// TwinCAT 3 PLC project ServerMappingSampleProject_PLC2
// Title: TF6100_OpcUa_Server_Sample_PLC2
// Company: Beckhoff Automation Gmbh
// ProjectVersion: 0.0.0.0
// ProgramVersion: 3.1.4026.17
// libraries:
//   Tc2_Standard, * (Beckhoff Automation GmbH)
//   Tc2_System, * (Beckhoff Automation GmbH)
// project tree:
//   / PlcTask.TcTTO
//   POUs/ MAIN.TcPOU
// (motion and I/O tree: see PLC project servermappingsampleproject)
// real-time tasks:
//   TASK Task1: cycle T#10ms, priority 20, ADS port 350
//   TASK Task2: cycle T#10ms, priority 21, ADS port 351
//   TASK PlcTask: cycle T#10ms, priority 22, ADS port 352

CONFIGURATION ServerMappingSampleProject_PLC2
    RESOURCE PLC ON TwinCAT3
        TASK PlcTask(INTERVAL := T#10ms, PRIORITY := 22);
        PROGRAM MAIN WITH PlcTask : MAIN;
    END_RESOURCE
END_CONFIGURATION

// ---- POUs/MAIN.TcPOU
PROGRAM MAIN
VAR
	//From this PLC only simple types can be mapped, because tmc is not enabled. 
	//For complex types and methods to work, tmc would need to be enabled. 
	//Also the DA-Config from the server would need this plc to be configured for the tmc to be loaded upon startup.
	
	bBoolFromSecondsAdsDevice : BOOL;// Boolean variable toggling based on timer
    fbTon : TON; // Timer function block
END_VAR

// Timer settings: 500 milliseconds time delay
fbTon(IN:= TRUE, PT:= T#500ms);

// Toggle logic
IF fbTon.Q THEN
    bBoolFromSecondsAdsDevice := NOT bBoolFromSecondsAdsDevice;
    fbTon(IN:= FALSE); // Reset the timer
END_IF

// Restart the timer
IF NOT fbTon.IN THEN
    fbTon(IN:= TRUE);
END_IF

END_PROGRAM
